// TIA Portal project "S7-1500 Analog Giriş ile Su Deposu" (V18)

(* hardware
DEVICE "S7-1500/ET200MP station_1"  S7-1500 station
   slot 0: "Rail_0"  Rack  6ES7 590-1***0-0AA0
   slot 1: "PLC_1"  CPU 1512C-1 PN  6ES7 512-1CK01-0AB0  V2.8
      slot 3: "CPU display_1"  6ES7591-1AA00-0AA0
      slot 32768: "PROFINET interface_1"  X1
         slot 32769: "Port_1"  X1 P1
         slot 32770: "Port_2"  X1 P2
      slot 34817: "Virtual CP interface port_1"  Virtual CP interface port  Virtual CP interface port
DEVICE "HMI_1"  KTP700 Basic PN
   slot 0: "HMI_1"  KTP700 Basic PN  6AV2 123-2GB03-0AX0  14.0.1.0
   slot 1: "HMI_RT_1"  KTP700 Basic PN  6AV2 123-2GB03-0AX0  14.0.1.0
   slot 5: "HMI_1.IE_CP_1"  PROFINET Interface  14.0.1.0
      slot 1: "PROFINET Interface_1"  PROFINET Interface
         slot 1: "Port_1"  Port
*)

// ===== PLC "PLC_1"  CPU 1512C-1 PN =====

VAR_GLOBAL   // PLC tag table "Default tag table"
   "Analog Giriş" AT %IW126 : Word;
   "Analog Yardımcı" AT %MW126 : Word;
   "sayaç_1" AT %MD10 : DWord;
   "sayaç_2" AT %MW20 : Int;
   "Doldurma Motoru_1" AT %Q0.1 : Bool;
   "Doldurma Motoru_2" AT %Q0.2 : Bool;
   "Tahliye Motoru" AT %Q0.3 : Bool;
END_VAR

ORGANIZATION_BLOCK "Main"   // OB1, LAD, ProgramCycle
TITLE = "Main Program Sweep (Cycle)"
{ S7_Optimized_Access := 'TRUE' }
VERSION : 0.1
   VAR_INPUT
      Initial_Call : Bool;   // Initial call of this OB
      Remanence : Bool;   // =True, if remanent data are available
   END_VAR
   VAR_TEMP   // added for the SCL form of the ladder/FBD networks
      _w1 : Bool;
   END_VAR
BEGIN

REGION Network 1: Analog girişten alınan değeri okumak içindir.
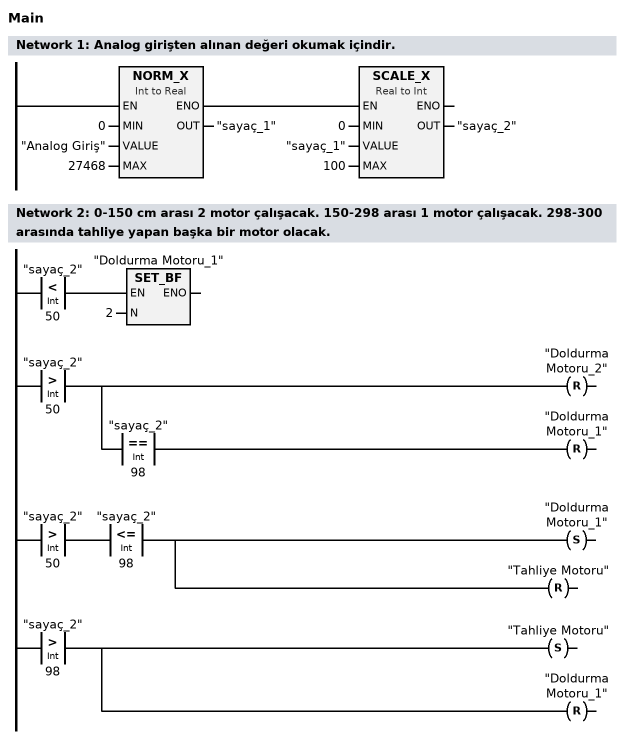
   RUNG wire#powerrail
      { S7_Templates := "[SrcType := Int, DestType := Real]" } Normalize(min := 0, value := "Analog Giriş", max := 27468, out => "sayaç_1")
      { S7_Templates := "[SrcType := Real, DestType := Int]" } Scale(min := 0, value := "sayaç_1", max := 100, out => "sayaç_2")
   END_RUNG
   // the same network as SCL:
   "sayaç_1" := NORM_X(MIN := 0, VALUE := "Analog Giriş", MAX := 27468);
   "sayaç_2" := SCALE_X(MIN := 0, VALUE := "sayaç_1", MAX := 100);
END_REGION

REGION Network 2: 0-150 cm arası 2 motor çalışacak. 150-298 arası 1 motor çalışacak. 298-300 arasında tahliye yapan başka bir motor olacak.
   // no SCL statement known for SBitfield: written as a call
   IF "sayaç_2" < 50 THEN SET_BF(operand := "Doldurma Motoru_1", n := 2); END_IF;
   #_w1 := "sayaç_2" > 50;
   IF #_w1 THEN "Doldurma Motoru_2" := FALSE; END_IF;
   IF #_w1 AND ("sayaç_2" = 98) THEN "Doldurma Motoru_1" := FALSE; END_IF;
   IF ("sayaç_2" > 50) AND ("sayaç_2" <= 98) THEN
       "Doldurma Motoru_1" := TRUE;
       "Tahliye Motoru" := FALSE;
   END_IF;
   IF "sayaç_2" > 98 THEN
       "Tahliye Motoru" := TRUE;
       "Doldurma Motoru_1" := FALSE;
   END_IF;
END_REGION
END_ORGANIZATION_BLOCK

(* ===== HMI "HMI_RT_1" =====
system functions are stored by id; their names below are inferred from use
connection "Connection_1": ETHERNET, SMART_S7_1500_OMS
connection "HMI_Connection_1": ETHERNET, SMART_S7_1500_OMS

HMI tags "Default tag table"
   "Tag_ScreenNumber" : UInt, internal
   "sayaç_2" : Int = PLC sayaç_2 AT %MW20, 100 ms
   "Doldurma Motoru_1" : Bool = PLC "Doldurma Motoru_1" AT %Q0.1, 100 ms
   "Doldurma Motoru_2" : Bool = PLC "Doldurma Motoru_2" AT %Q0.2, 100 ms
   "Tahliye Motoru" : Bool = PLC "Tahliye Motoru" AT %Q0.3, 100 ms

graphic list "Motor_1": 0 'Graphic_13'; 1 'Graphic_12'

graphic list "Motor_2": 0 'Graphic_10'; 1 'Graphic_11'

graphic list "Taziye Musluğu": 0 'Graphic_6'; 1 'Graphic_7'

Template "Template_1" 800x480
   Button "Exit" at 714,429 size 71x50; TextOff 'Exit'; PictureOff "ExitRuntime_KTP700_Basic_PN_TR"; PictureOn "ExitRuntime_KTP700_Basic_PN_TR"
      on Release: StopRuntime(0)
   Button "Language" at 614,429 size 71x50; TextOff 'Language'; PictureOff "ToggleLanguage_KTP700_Basic_PN_TR"; PictureOn "ToggleLanguage_KTP700_Basic_PN_TR"
      on Release: function_fb9197e8(-1)
   Button "Log on" at 514,429 size 71x50; TextOff 'Log on'; PictureOff "Login_KTP700_Basic_PN_TR"; PictureOn "Login_KTP700_Basic_PN_TR"
      on Release: function_a2a04561()
   Button "Alarms" at 114,429 size 71x50; TextOff 'Alarms'; PictureOff "AlarmDisplay_KTP700_Basic_PN_TR"; PictureOn "AlarmDisplay_KTP700_Basic_PN_TR"
      on Release: function_ef3f5d25("Alarm window_Unacknowledged", -1)
   Button "Start screen" at 14,429 size 71x50; TextOff 'Start screen'; PictureOff "NavigateHome_KTP700_Basic_PN_TR"; PictureOn "NavigateHome_KTP700_Basic_PN_TR"
      on Release: ActivateScreen("Root screen", 0)
   SymbolicIOField "Symbolic_IO_Field_Screen" at 93,9 size 600x33; TextOff '0'; TextOn '1'; TextList "TextList_ScreenNames"
      ProcessValue <- "Tag_ScreenNumber"
      on Change: ActivateScreenByNumber("Tag_ScreenNumber", 0)
   DateTimeField "HmiScreenItemData" at 695,25 size 105x25
   DateTimeField "HmiScreenItemData_1" at 695,0 size 105x25
   GraphicView "Logo" at 0,0 size 91x51; Picture "Logo of HMI_1"

screen "Root screen" 800x480, template "Template_1"
   on GenerateScreen: SetTag("Tag_ScreenNumber", 1)
   Bar "Bar_1" at 394,88 size 134x240; MinimumValue 0; MaximumValue 100
      ProcessValue <- "sayaç_2"
   GraphicIOField "Graphic I/O field_1" at 410,327 size 96x48; PictureList "Taziye Musluğu"
      ProcessValue <- "Tahliye Motoru"
   GraphicIOField "Graphic I/O field_2" at 528,181 size 96x48; PictureList "Motor_2"
      ProcessValue <- "Doldurma Motoru_2"
   GraphicIOField "Graphic I/O field_3" at 298,88 size 96x48; PictureList "Motor_1"
      ProcessValue <- "Doldurma Motoru_1"
   IOField "I/O field_1" at 254,180 size 117x78; FormatPattern s99999
      ProcessValue <- "sayaç_2"
*)